FUNCTION Convert_BYTE_TO_UINT : Hresult
VAR_INPUT
	in : BYTE;
	out : REFERENCE TO UINT;
END_VAR
VAR
	converted : UINT;
END_VAR
VAR CONSTANT
	INCOMPATIBLE : HRESULT := 16#9811070E;
END_VAR

converted := BYTE_TO_UINT(in);

IF (UINT_TO_BYTE(converted) <> in) THEN
	Convert_BYTE_TO_UINT := INCOMPATIBLE;
	RETURN;
END_IF

out := converted;

END_FUNCTION

(* stored: Version 1.1.0.1, ProductVersion 3.1.4024.12
   POU Convert_BYTE_TO_UINT: Id {d2246b57-5ae6-4c25-83f5-9a468a6fe159}, SpecialFunc None *)
